(* IEC 61131-3 sources: RL_MAR/experiments/comparison/llm4plc/results/gpt-4o_20260507_114630/20260507_120247, 1 file *)

(* ---- generated_code_iteration_0.st ---- *)
plaintext
START_ST
FUNCTION_BLOCK SandwichMaker
VAR_INPUT
    BreadFeeder : BOOL; (* Input: Detects the presence of bread slices *)
    Ingredient1 : BOOL; (* Input: Detects the presence of Ingredient 1 (e.g., cheese) *)
    Ingredient2 : BOOL; (* Input: Detects the presence of Ingredient 2 (e.g., lettuce) *)
    Ingredient3 : BOOL; (* Input: Detects the presence of Ingredient 3 (e.g., tomatoes) *)
    Condiment1 : BOOL; (* Input: Detects the presence of Condiment 1 (e.g., mayo) *)
    Condiment2 : BOOL; (* Input: Detects the presence of Condiment 2 (e.g., mustard) *)
END_VAR
VAR_OUTPUT
    ConveyorMotor : BOOL; (* Output: Controls the conveyor belt motor *)
    AssembleMotor : BOOL; (* Output: Controls the sandwich assembly motor *)
END_VAR
VAR
    state : INT := 0; (* The current state of the system *)
    prevState : INT := 0; (* The previous state of the system *)
    SliceCount : INT := 0; (* Counter for bread slices *)
END_VAR

(* State Definitions *)
(* STATE 0: IDLE *)
(* STATE 1: DETECT_BREAD *)
(* STATE 2: CHECK_INGREDIENTS *)
(* STATE 3: ASSEMBLE_SANDWICH *)

(* Main Logic *)
CASE state OF
    0: (* IDLE *)
        ConveyorMotor := FALSE; (* Conveyor motor is off *)
        AssembleMotor := FALSE; (* Assembly motor is off *)
        IF BreadFeeder THEN
            state := 1; (* Transition to DETECT_BREAD state *)
        END_IF;

    1: (* DETECT_BREAD *)
        ConveyorMotor := TRUE; (* Conveyor motor is on *)
        AssembleMotor := FALSE; (* Assembly motor is off *)
        IF BreadFeeder THEN
            SliceCount := SliceCount + 1; (* Increment slice count *)
        END_IF;
        IF SliceCount >= 2 THEN
            state := 2; (* Transition to CHECK_INGREDIENTS state *)
        END_IF;

    2: (* CHECK_INGREDIENTS *)
        ConveyorMotor := FALSE; (* Conveyor motor is off *)
        AssembleMotor := FALSE; (* Assembly motor is off *)
        IF Ingredient1 AND Ingredient2 AND Ingredient3 AND Condiment1 AND Condiment2 THEN
            state := 3; (* Transition to ASSEMBLE_SANDWICH state *)
        ELSIF NOT BreadFeeder OR SliceCount < 2 OR NOT (Ingredient1 AND Ingredient2 AND Ingredient3 AND Condiment1 AND Condiment2) THEN
            state := 0; (* Transition back to IDLE state *)
        END_IF;

    3: (* ASSEMBLE_SANDWICH *)
        ConveyorMotor := FALSE; (* Conveyor motor is off *)
        AssembleMotor := TRUE; (* Assembly motor is on *)
        IF NOT BreadFeeder THEN
            state := 0; (* Transition back to IDLE state *)
        END_IF;

    ELSE
        (* Default case to handle unexpected states *)
        state := 0; (* Reset to IDLE state *)
END_CASE;

END_FUNCTION_BLOCK
END_ST
